PROGRAM MAIN
VAR
	ObranPoczatkowy:FB_Glowny;
	gra:FB_Snake;
END_VAR

ObranPoczatkowy();
gra();

END_PROGRAM

(* stored: Version 1.1.0.1, ProductVersion 3.1.4024.4
   POU MAIN: Id {003304d9-0937-481e-94b7-806557916c6d}, SpecialFunc None *)
